// TIA Portal project "SpringControl" (V18)

(* hardware
DEVICE "S7-1500/ET200MP station_1"  S7-1500 station
   slot 0: "PM 190W 120/230VAC"  PM 190W 120/230VAC  6EP1333-4BA00
   slot 0: "导轨_0"  Rack  6ES7 590-1***0-0AA0
   slot 1: "PLC_1"  CPU 1511-1 PN  6ES7 511-1AK02-0AB0  V2.9
      slot 3: "CPU 显示_1"  6ES7591-1AA00-0AA0
      slot 32768: "PROFINET 接口_1"  X1
         slot 32769: "端口_1"  X1 P1
         slot 32770: "端口_2"  X1 P2
      slot 34817: "Virtual CP interface port_1"  Virtual CP interface port  Virtual CP interface port
   slot 2: "DI 16x24VDC HF_1"  DI 16x24VDC HF  6ES7 521-1BH00-0AB0  V2.2
   slot 3: "DQ 16x24VDC/0.5A HF_1"  DQ 16x24VDC/0.5A HF  6ES7 522-1BH01-0AB0  V1.1
   slot 4: "AI 8xU/I/RTD/TC ST_1"  AI 8xU/I/RTD/TC ST  6ES7 531-7KF00-0AB0  V2.2
   slot 5: "AQ 4xU/I ST_1"  AQ 4xU/I ST  6ES7 532-5HD00-0AB0  V2.2
*)

// ===== PLC "PLC_1"  CPU 1511-1 PN =====

VAR_GLOBAL   // PLC tag table "默认变量表"
   "System_Byte" AT %MB1000 : Byte;
   "FirstScan" AT %M1000.0 : Bool;
   "DiagStatusUpdate" AT %M1000.1 : Bool;
   "AlwaysTRUE" AT %M1000.2 : Bool;
   "AlwaysFALSE" AT %M1000.3 : Bool;
   "Clock_Byte" AT %MB1001 : Byte;
   "Clock_10Hz" AT %M1001.0 : Bool;
   "Clock_5Hz" AT %M1001.1 : Bool;
   "Clock_2.5Hz" AT %M1001.2 : Bool;
   "Clock_2Hz" AT %M1001.3 : Bool;
   "Clock_1.25Hz" AT %M1001.4 : Bool;
   "Clock_1Hz" AT %M1001.5 : Bool;
   "Clock_0.625Hz" AT %M1001.6 : Bool;
   "Clock_0.5Hz" AT %M1001.7 : Bool;
   "Tag_1" AT %M0.1 : Bool;
END_VAR

VAR_GLOBAL   // PLC tag table "物理变量表"
   "SB1" AT %I0.0 : Bool;
   "SB2" AT %I0.1 : Bool;
   "P1" AT %Q4.0 : Bool;
   "P2" AT %Q4.1 : Bool;
   "A1" AT %Q5.0 : Bool;
   "A2" AT %Q5.1 : Bool;
   "A3" AT %Q5.2 : Bool;
   "A4" AT %Q5.3 : Bool;
   "A5" AT %Q5.4 : Bool;
   "A6" AT %Q5.5 : Bool;
   "B1" AT %Q6.0 : Bool;
   "B2" AT %Q6.1 : Bool;
   "B3" AT %Q6.2 : Bool;
   "B4" AT %Q6.3 : Bool;
   "B5" AT %Q6.4 : Bool;
   "B6" AT %Q6.5 : Bool;
END_VAR

DATA_BLOCK "sj"   // DB2
{ S7_Optimized_Access := 'TRUE' }
VERSION : 0.1
   VAR
      Overall : Bool;
      State0 : Bool := true;
      State1 : Bool;
      State2 : Bool;
      State3 : Bool;
   END_VAR
BEGIN
END_DATA_BLOCK

// folder: System blocks/Program resources

DATA_BLOCK "IEC_Timer_0_DB"   // DB1
{ S7_Optimized_Access := 'TRUE' }
AUTHOR : Simatic
FAMILY : IEC
NAME : IEC_TMR
VERSION : 1.0
// stored: InstanceOfName IEC_TIMER
"IEC_TIMER"
BEGIN
END_DATA_BLOCK

DATA_BLOCK "IEC_Timer_0_DB_1"   // DB3
{ S7_Optimized_Access := 'TRUE' }
AUTHOR : Simatic
FAMILY : IEC
NAME : IEC_TMR
VERSION : 1.0
// stored: InstanceOfName IEC_TIMER
"IEC_TIMER"
BEGIN
END_DATA_BLOCK

DATA_BLOCK "IEC_Timer_0_DB_2"   // DB4
{ S7_Optimized_Access := 'TRUE' }
AUTHOR : Simatic
FAMILY : IEC
NAME : IEC_TMR
VERSION : 1.0
// stored: InstanceOfName IEC_TIMER
"IEC_TIMER"
BEGIN
END_DATA_BLOCK

DATA_BLOCK "IEC_Timer_0_DB_3"   // DB5
{ S7_Optimized_Access := 'TRUE' }
AUTHOR : Simatic
FAMILY : IEC
NAME : IEC_TMR
VERSION : 1.0
// stored: InstanceOfName IEC_TIMER
"IEC_TIMER"
BEGIN
END_DATA_BLOCK

DATA_BLOCK "IEC_Timer_0_DB_4"   // DB6
{ S7_Optimized_Access := 'TRUE' }
AUTHOR : Simatic
FAMILY : IEC
NAME : IEC_TMR
VERSION : 1.0
// stored: InstanceOfName IEC_TIMER
"IEC_TIMER"
BEGIN
END_DATA_BLOCK

// folder: (top level)

FUNCTION_BLOCK "定时器"   // FB1, LAD
{ S7_Optimized_Access := 'TRUE' }
VERSION : 0.1
   VAR_INPUT
      Timing : Time;
      NowState : Bool;
   END_VAR
   VAR_OUTPUT
      SetNextState : Bool;
      ResetNowState : Bool;
   END_VAR
BEGIN

REGION Network 1
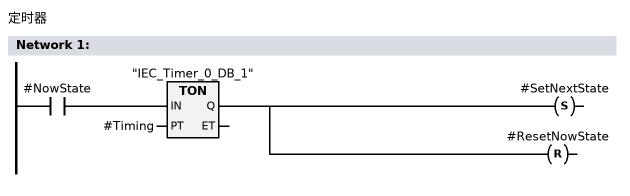
   "IEC_Timer_0_DB_1".TON(IN := #NowState, PT := #Timing);
   IF "IEC_Timer_0_DB_1".Q THEN
       #SetNextState := TRUE;
       #ResetNowState := FALSE;
   END_IF;
END_REGION
END_FUNCTION_BLOCK

ORGANIZATION_BLOCK "Main"   // OB1, LAD, ProgramCycle
TITLE = "Main Program Sweep (Cycle)"
{ S7_Optimized_Access := 'TRUE' }
VERSION : 0.1
   VAR_INPUT
      Initial_Call : Bool;   // Initial call of this OB
      Remanence : Bool;   // =True, if remanent data are available
   END_VAR
   VAR CONSTANT
      ll : Bool := true;
   END_VAR
   VAR_TEMP   // added for the SCL form of the ladder/FBD networks
      _w1 : Bool;
      _w2 : Bool;
   END_VAR
BEGIN

REGION Network 1: PowerControl
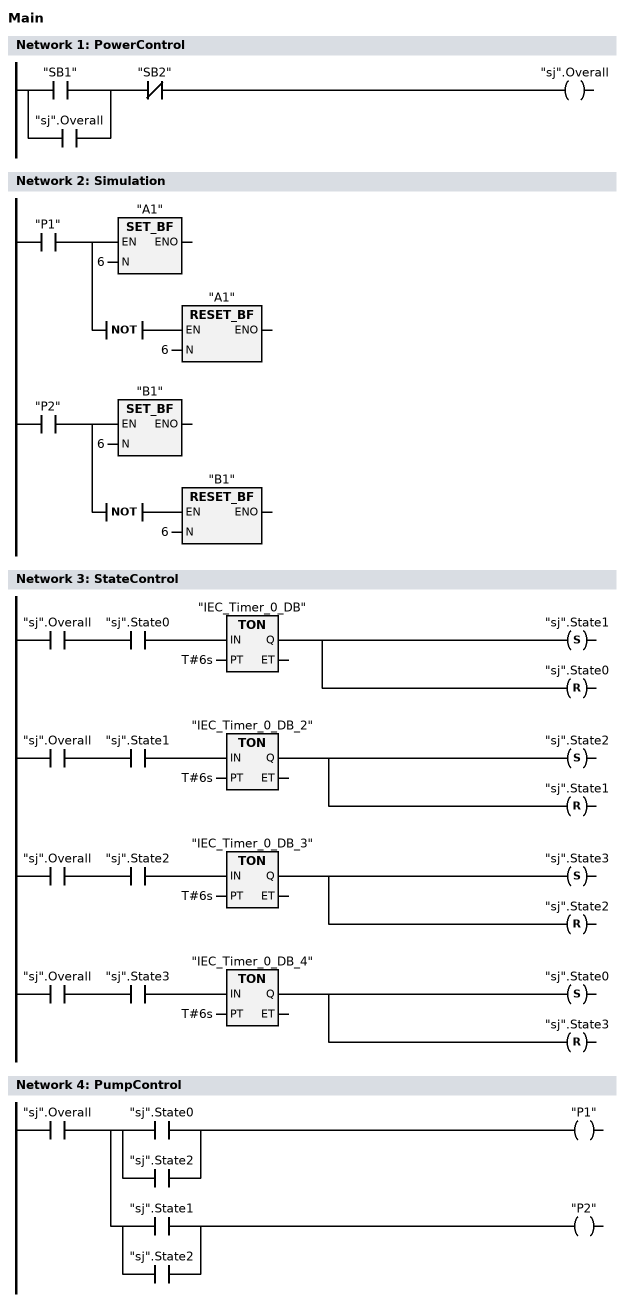
   RUNG wire#powerrail
      Contact( "SB1" )
      wire#w1
      I_Contact( "SB2" )
      Coil( "sj".Overall )
   END_RUNG
   RUNG wire#powerrail
      Contact( "sj".Overall )
   END_RUNG wire#w1
   // the same network as SCL:
   "sj".Overall := ("SB1" OR "sj".Overall) AND NOT "SB2";
END_REGION

REGION Network 2: Simulation
   // no SCL statement known for RBitfield, SBitfield: written as a call
   #_w1 := "P1";
   IF #_w1 THEN SET_BF(operand := "A1", n := 6); END_IF;
   IF NOT #_w1 THEN RESET_BF(operand := "A1", n := 6); END_IF;
   #_w2 := "P2";
   IF #_w2 THEN SET_BF(operand := "B1", n := 6); END_IF;
   IF NOT #_w2 THEN RESET_BF(operand := "B1", n := 6); END_IF;
END_REGION

REGION Network 3: StateControl
   "IEC_Timer_0_DB".TON(IN := "sj".Overall AND "sj".State0, PT := T#6s);
   IF "IEC_Timer_0_DB".Q THEN
       "sj".State1 := TRUE;
       "sj".State0 := FALSE;
   END_IF;
   "IEC_Timer_0_DB_2".TON(IN := "sj".Overall AND "sj".State1, PT := T#6s);
   IF "IEC_Timer_0_DB_2".Q THEN
       "sj".State2 := TRUE;
       "sj".State1 := FALSE;
   END_IF;
   "IEC_Timer_0_DB_3".TON(IN := "sj".Overall AND "sj".State2, PT := T#6s);
   IF "IEC_Timer_0_DB_3".Q THEN
       "sj".State3 := TRUE;
       "sj".State2 := FALSE;
   END_IF;
   "IEC_Timer_0_DB_4".TON(IN := "sj".Overall AND "sj".State3, PT := T#6s);
   IF "IEC_Timer_0_DB_4".Q THEN
       "sj".State0 := TRUE;
       "sj".State3 := FALSE;
   END_IF;
END_REGION

REGION Network 4: PumpControl
   RUNG wire#powerrail
      Contact( "sj".Overall )
      wire#w1
      Contact( "sj".State0 )
      wire#w2
      Coil( "P1" )
   END_RUNG
   RUNG wire#w1
      Contact( "sj".State2 )
   END_RUNG wire#w2
   RUNG wire#w1
      Contact( "sj".State1 )
      wire#w3
      Coil( "P2" )
   END_RUNG
   RUNG wire#w1
      Contact( "sj".State2 )
   END_RUNG wire#w3
   // the same network as SCL:
   "P1" := "sj".Overall AND ("sj".State0 OR "sj".State2);
   "P2" := "sj".Overall AND ("sj".State1 OR "sj".State2);
END_REGION
END_ORGANIZATION_BLOCK